{attribute 'GeneratedUsingTerminal: EP7402-0057-0017'}
{attribute addProperty BoxType "EP7402-0057-0017"}
{attribute addProperty Id "A_0055_EP7402_0057_0018EP7402_E132E05C99"}
{attribute addProperty CRC "1368330331"}
{attribute addProperty Size "99"}
TYPE A_0054_EP7402_0057_0017_518F105B EXTENDS EP7402_E132E05C :
STRUCT
	{attribute addProperty Name "A_0055_EP7402_0057_0018"}
	{attribute addProperty PreviousPort "A_0054(EP7402-0057-0017) : B"}
	A_0055_EP7402_0057_0018 : EP7402_E132E05C;
END_STRUCT
END_TYPE

(* stored: Version 1.2.0.0, ProductVersion 3.1.4024.9
   DUT A_0054_EP7402_0057_0017_518F105B: Id {6549206b-89ae-44ef-a41c-e2969286e879} *)
